Universal Robots URScript: 20240827calipoint.script

def P20240827calipoint():
  global _hidden_verificationVariable=0
  set_safety_mode_transition_hardness(0)
  set_target_payload(1.500000, [0.001000, -0.003000, 0.050000], [0.003026, 0.003026, 0.003026, 0.000000, 0.000000, 0.000000])
  set_gravity([0.0, 0.0, 9.82])
  set_tcp(p[-1.7E-4,0.0,0.19294999999999998,0.0,0.0,0.0])
  set_standard_analog_input_domain(0, 1)
  set_standard_analog_input_domain(1, 1)
  set_tool_analog_input_domain(0, 1)
  set_tool_analog_input_domain(1, 1)
  set_analog_outputdomain(0, 1)
  set_analog_outputdomain(1, 0)
  set_input_actions_to_default()
  set_tool_digital_input_action(0, "freedrive")
  set_tool_communication(True, 115200, 0, 1, 1.5, 3.5)
  set_tool_output_mode(0)
  set_tool_digital_output_mode(0, 1)
  set_tool_digital_output_mode(1, 1)
  set_tool_voltage(24)
  global i_var_1=p[0.31, 0, 0, 0, 0, 0]
  global u24179u38754_1=p[0.0,0.0,0.0,0.0,0.0,0.0]
  global u24179u38754_2=p[0.2,0.6,0.4,-1.4839444017850547,-0.07419722008925289,-2.225916602677581]
  global u24179u38754_3=p[0.1459477485431481,-0.10308445883660293,0.13857682671027435,-0.008977024873201634,0.014216906208388691,-2.4400986907073663]
  global u28857_1=p[0.10203918836050063,-0.5259531579406657,0.376430278847906,-0.18768520041296463,-3.1325095402283982,-0.09669790600413578]
  global u28857_2=p[0.0665007526844362,-0.3872123180436422,0.638459113340625,-0.320095108678139,-2.6903368475934015,1.4700117755369673]
  global u30452u32447_1=p[0.0,0.0,0.0,0.0,0.0,0.0]
  step_count_1a284065_73db_4a87_86ac_5485ac17be38 = 0.0
  thread Step_Counter_Thread_03664bf6_442c_4511_b66b_bd81e107a8a9():
    while (True):
      step_count_1a284065_73db_4a87_86ac_5485ac17be38 = step_count_1a284065_73db_4a87_86ac_5485ac17be38 + 1.0
      sync()
    end
  end
  run Step_Counter_Thread_03664bf6_442c_4511_b66b_bd81e107a8a9()
  global photo_p=p[.096736129787, -.476129287342, .310081590554, -1.949365627478, -1.826188223498, -.604869100606]
  global photo_q=[1.4917473793029785, -1.4001578849605103, 1.746774975453512, -1.3199018400958558, -1.5736311117755335, 1.5610498189926147]
  global u36335u28857_1_p=p[.093501898871, -.542216259301, -.001231601139, 2.051451198771, 1.923945434942, -.388364666693]
  global u36335u28857_1_q=[1.4504916667938232, -1.766609331170553, 2.377599064503805, -2.063395162621969, -1.5448325316058558, 1.506522536277771]
  global u36335u28857_2_p=p[.093498408578, -.542195933642, -.001248842075, 2.094517114891, 2.120621806814, -.813264363106]
  global u36335u28857_2_q=[1.7910959720611572, -1.597640176812643, 2.283836905156271, -2.0663486919798792, -1.8604334036456507, 1.8979114294052124]
  global u36335u28857_3_p=p[.093497390241, -.542220936525, -.001231164968, -1.855813354258, -2.079353441855, .650639515634]
  global u36335u28857_3_q=[1.8728539943695068, -1.3699295085719605, 1.8873966375934046, -1.5252489385059853, -1.9388883749591272, 2.0128228664398193]
  global u36335u28857_4_p=p[.093516021533, -.542183369037, -.001265484308, -1.677058249824, -2.000050144554, .455645328932]
  global u36335u28857_4_q=[1.879108190536499, -1.171933875685074, 1.5747621695147913, -1.1577239793590088, -1.9384163061725062, 2.0304229259490967]
  global u36335u28857_5_p=p[.093513394102, -.542219718617, -.001238047151, -1.477844903041, -2.035523293769, -.083831770926]
  global u36335u28857_5_q=[1.7509469985961914, -0.8956406873515625, 1.0779522101031702, -0.6746114057353516, -1.9029443899737757, 1.7342504262924194]
  global u36335u28857_6_p=p[.093490285155, -.542201139551, -.001233373493, -1.478437948851, -2.248857168536, -.459269446984]
  global u36335u28857_6_q=[1.5786175727844238, -0.9081941407969971, 1.0524728933917444, -0.690642313366272, -1.8782098929034632, 1.3333466053009033]
  global u36335u28857_7_p=p[.093511148404, -.542223662535, -.001237021723, -1.502345725756, -2.514544997169, -.718639272788]
  global u36335u28857_7_q=[1.4066588878631592, -0.9898206156543274, 1.2026165167437952, -0.8718646925738831, -1.8344939390765589, 0.9467003345489502]
  global u36335u28857_8_p=p[.093520703009, -.542225368445, -.001245345625, -1.468768578600, -2.534521422812, -1.080282010409]
  global u36335u28857_8_q=[1.319551944732666, -0.8169216078570862, 1.0130322615252894, -0.7210088533214112, -1.7973583380328577, 0.7572055459022522]
  global u36335u28857_9_p=p[.093506434033, -.542217913664, -.001223102207, 1.373437457907, 2.524760477293, .924188910839]
  global u36335u28857_9_q=[1.262399435043335, -0.9633787435344239, 1.254549805318014, -0.9641900223544617, -1.7734978834735315, 0.6178150177001953]
  global u36335u28857_10_p=p[.093517903476, -.542202351315, -.001241077192, 1.319460153553, 2.630225971412, .309326938139]
  global u36335u28857_10_q=[1.2716752290725708, -1.3604417604259034, 1.7805026213275355, -1.513977364902832, -1.7879293600665491, 0.6151435375213623]
  global u36335u28857_11_p=p[.093505734071, -.542224359274, -.001232364858, 1.198218947526, 2.480808161758, .041572612542]
  global u36335u28857_11_q=[1.132570505142212, -1.5274053190699597, 2.105126682912008, -1.899297376672262, -1.6602070967303675, 0.42513346672058105]
  global u36335u28857_12_p=p[.093511150298, -.542189105023, -.001268356415, 1.217911110830, 2.651905081760, -.197166205830]
  global u36335u28857_12_q=[1.286444067955017, -1.6226893864073695, 2.1781943480121058, -2.001136919061178, -1.8132689634906214, 0.6028025150299072]
  global u36335u28857_13_p=p[.093505961011, -.542184044579, -.001265214391, 1.225397892035, 2.842860972139, -.503341719311]
  global u36335u28857_13_q=[1.5183889865875244, -1.6545163593687953, 2.227274719868795, -2.057315012017721, -2.0452397505389612, 0.862866222858429]
  global u36335u28857_14_p=p[.093505940171, -.542214284748, -.001232431736, -1.124606598719, -2.692614035751, .412865554950]
  global u36335u28857_14_q=[1.6652103662490845, -1.5277397495559235, 2.0201028029071253, -1.7429434261717738, -2.1760600248919886, 1.080268144607544]
  global u36335u28857_15_p=p[.093485281750, -.542214535278, -.001227720539, -1.340511871148, -2.429475958723, .407755398373]
  global u36335u28857_15_q=[1.7814942598342896, -1.3891225916198273, 1.8291376272784632, -1.420476273899414, -2.125793759022848, 1.5106902122497559]
  global u36335u28857_16_p=p[.093502505368, -.542179875077, -.001251475903, -1.524179520451, -2.163660510999, .250138253446]
  global u36335u28857_16_q=[1.8060213327407837, -1.171669678097107, 1.510975186024801, -1.0738120538047333, -1.9816601912127894, 1.7732305526733398]
  global u36335u28857_17_p=p[.093508579661, -.542197641026, -.001238433578, -2.014439072175, -1.804873652858, .054280707616]
  global u36335u28857_17_q=[1.7077686786651611, -1.0870579046062012, 1.3470199743853968, -0.9816933435252686, -1.6612055937396448, 1.9610741138458252]
  global u36335u28857_18_p=p[.093514578462, -.542190956199, -.001243127379, -2.160546416548, -1.509146290037, -.124413837021]
  global u36335u28857_18_q=[1.6484122276306152, -0.9366257947734375, 1.116795841847555, -0.803161696796753, -1.4905126730548304, 2.0661182403564453]
  global u36335u28857_19_p=p[.093514351783, -.542214372774, -.001242083604, -2.431458256377, -1.316591791321, -.522300300669]
  global u36335u28857_19_q=[1.4471406936645508, -0.9807250064662476, 1.164382282887594, -0.7744110983661194, -1.2660883108722132, 1.8991031646728516]
  global u36335u28857_20_p=p[.093495008382, -.542232265117, -.001215767680, -2.291881618246, -1.820213941595, -.574321542072]
  global u36335u28857_20_q=[1.3973069190979004, -1.1048370164683838, 1.3386614958392542, -0.8796340388110657, -1.4390767256366175, 1.5305410623550415]
  def takephoto():
    $ 54 "takephoto" "noBreak"
    $ 55 "等待: 1.0"
    sleep(1.0)
    $ 56 "cam.takePhoto(get_actual_tcp_pose())"
    cam.takePhoto( get_actual_tcp_pose ())
    $ 57 "弹出窗口: please ensure "
    popup("please ensure ", "消息", False, False, blocking=True)
  end
  $ 2 "机器人程序"
  $ 3 "cam≔rpc_factory('xmlrpc', 'http://192.168.1.5:9130/RPC2')"
  global cam=rpc_factory("xmlrpc", "http://192.168.1.5:9130/RPC2")
  $ 5 "MoveJ"
  $ 6 "photo" "breakAfter"
  movej(photo_q, a=1.3962634015954636, v=1.0471975511965976)
  $ 7 "调用 takephoto"
  takephoto()
  $ 9 "MoveJ"
  $ 10 "路点_1" "breakAfter"
  movej(u36335u28857_1_q, a=1.3962634015954636, v=1.0471975511965976)
  $ 11 "调用 takephoto"
  takephoto()
  $ 12 "路点_2" "breakAfter"
  movej(u36335u28857_2_q, a=1.3962634015954636, v=1.0471975511965976)
  $ 13 "调用 takephoto"
  takephoto()
  $ 14 "路点_3" "breakAfter"
  movej(u36335u28857_3_q, a=1.3962634015954636, v=1.0471975511965976)
  $ 15 "调用 takephoto"
  takephoto()
  $ 16 "路点_4" "breakAfter"
  movej(u36335u28857_4_q, a=1.3962634015954636, v=1.0471975511965976)
  $ 17 "调用 takephoto"
  takephoto()
  $ 18 "路点_5" "breakAfter"
  movej(u36335u28857_5_q, a=1.3962634015954636, v=1.0471975511965976)
  $ 19 "调用 takephoto"
  takephoto()
  $ 20 "路点_6" "breakAfter"
  movej(u36335u28857_6_q, a=1.3962634015954636, v=1.0471975511965976)
  $ 21 "调用 takephoto"
  takephoto()
  $ 22 "路点_7" "breakAfter"
  movej(u36335u28857_7_q, a=1.3962634015954636, v=1.0471975511965976)
  $ 23 "调用 takephoto"
  takephoto()
  $ 24 "路点_8" "breakAfter"
  movej(u36335u28857_8_q, a=1.3962634015954636, v=1.0471975511965976)
  $ 25 "调用 takephoto"
  takephoto()
  $ 26 "路点_9" "breakAfter"
  movej(u36335u28857_9_q, a=1.3962634015954636, v=1.0471975511965976)
  $ 27 "调用 takephoto"
  takephoto()
  $ 28 "路点_10" "breakAfter"
  movej(u36335u28857_10_q, a=1.3962634015954636, v=1.0471975511965976)
  $ 29 "调用 takephoto"
  takephoto()
  $ 30 "路点_11" "breakAfter"
  movej(u36335u28857_11_q, a=1.3962634015954636, v=1.0471975511965976)
  $ 31 "调用 takephoto"
  takephoto()
  $ 32 "路点_12" "breakAfter"
  movej(u36335u28857_12_q, a=1.3962634015954636, v=1.0471975511965976)
  $ 33 "调用 takephoto"
  takephoto()
  $ 34 "路点_13" "breakAfter"
  movej(u36335u28857_13_q, a=1.3962634015954636, v=1.0471975511965976)
  $ 35 "调用 takephoto"
  takephoto()
  $ 36 "路点_14" "breakAfter"
  movej(u36335u28857_14_q, a=1.3962634015954636, v=1.0471975511965976)
  $ 37 "调用 takephoto"
  takephoto()
  $ 38 "路点_15" "breakAfter"
  movej(u36335u28857_15_q, a=1.3962634015954636, v=1.0471975511965976)
  $ 39 "调用 takephoto"
  takephoto()
  $ 40 "等待: 1.0"
  sleep(1.0)
  $ 41 "调用 takephoto"
  takephoto()
  $ 42 "路点_16" "breakAfter"
  movej(u36335u28857_16_q, a=1.3962634015954636, v=1.0471975511965976)
  $ 43 "调用 takephoto"
  takephoto()
  $ 44 "路点_17" "breakAfter"
  movej(u36335u28857_17_q, a=1.3962634015954636, v=1.0471975511965976)
  $ 45 "调用 takephoto"
  takephoto()
  $ 46 "路点_18" "breakAfter"
  movej(u36335u28857_18_q, a=1.3962634015954636, v=1.0471975511965976)
  $ 47 "调用 takephoto"
  takephoto()
  $ 48 "路点_19" "breakAfter"
  movej(u36335u28857_19_q, a=1.3962634015954636, v=1.0471975511965976)
  $ 49 "调用 takephoto"
  takephoto()
  $ 50 "路点_20" "breakAfter"
  movej(u36335u28857_20_q, a=1.3962634015954636, v=1.0471975511965976)
  $ 51 "调用 takephoto"
  takephoto()
  $ 52 "MoveJ"
  $ 53 "photo" "breakAfter"
  movej(photo_q, a=1.3962634015954636, v=1.0471975511965976)
end
